// TIA Portal V21 export
DATA_BLOCK "FlowMeter"   // DB28
{ S7_Optimized_Access := 'TRUE' }
// stored: MemoryReserve 100
   VAR
      FlowMeter : Array[0..1] of "Std_EthFlowMeter";
      PortataFM1 : Real := 0.0;
      PortataFM2 : Real := 190.2098;
   END_VAR
BEGIN
   // FlowMeter[0] : Decantazione -> Inspessitore
   // FlowMeter[1] : Decantazione -> Ossidazione
   FlowMeter[0].Volume_flow := 0.0;
   FlowMeter[1].Volume_flow := 190.2098;
   FlowMeter[0..1].Mass_Flow := 0.0;
   FlowMeter[0..1].Corrected_Volume_Flow := 0.0;
   FlowMeter[0..1].Velocity := 0.0;
   FlowMeter[0].Totalizer_1 := 0.0;
   FlowMeter[1].Totalizer_1 := 1285494.0;
   FlowMeter[0..1].Totalizer_2 := 0.0;
   FlowMeter[0..1].Totalizer_3 := 0.0;
   FlowMeter[0..1].ControlTotalizzatore_1 := 16#00;
   FlowMeter[0..1].ControlTotalizzatore_2 := 16#00;
   FlowMeter[0..1].ControlTotalizzatore_3 := 16#00;
END_DATA_BLOCK
